// TIA Portal project "TiaUnit" (V16)

(* hardware
DEVICE "S71500/ET200MP-Station_1"  S7-1500 station
   slot 0: "Profilschiene_0"  Rack  6ES7 590-1***0-0AA0
   slot 1: "PLC_1"  CPU 1513-1 PN  6ES7 513-1AL02-0AB0  V2.8
      slot 3: "CPU-Display_1"  6ES7591-1AA00-0AA0
      slot 32768: "PROFINET-Schnittstelle_1"  X1
         slot 32769: "Port_1"  X1 P1
         slot 32770: "Port_2"  X1 P2
      slot 34817: "Virtual CP interface port_1"  Virtual CP interface port  Virtual CP interface port
*)

// ===== PLC "PLC_1"  CPU 1513-1 PN =====

VAR_GLOBAL CONSTANT   // PLC tag table "Assert"
   "NOT_TESTED" : Byte := 16#00;
   "TEST_GOOD" : Byte := 16#01;
   "TEST_BAD" : Byte := 16#02;
END_VAR

TYPE "t_TIAUnit_Tests"
   STRUCT
      "step" : Word;
      result : Byte;
      text : String;
   END_STRUCT;
END_TYPE

TYPE "t_Assert"
   STRUCT
      testStart : Date_And_Time;
      testEnd : Date_And_Time;
      testGood : DInt;
      testBad : DInt;
      index : DInt;
      state : Word;
      stateMachineError : Bool;
   END_STRUCT;
END_TYPE

TYPE "t_AnalogInput"
   STRUCT
      PEW : DInt;   // Peripheral Input
      "Type" : UInt;
      SP1 : Bool;   // Switchpoint 1
      SP2 : Bool;   // Switchpoint 2
      SP3 : Bool;   // Switchpoint 3
      SP4 : Bool;   // Switchpoint 4
      SP5 : Bool;   // Switchpoint 5
      SP6 : Bool;   // Switchpoint 6
      SP7 : Bool;   // Switchpoint 7
      SP8 : Bool;   // Switchpoint 8
      CB : Bool;   // Cable break
      "OF" : Bool;   // Overflow
      SF : Bool;   // Sensor failure
      Bool3 : Bool;
      Bool4 : Bool;
      Bool5 : Bool;
      Bool6 : Bool;
      Bool7 : Bool;
      LoLim : Real := 0.0;   // Scaling Low-Limit
      HiLim : Real := 100.0;   // Scaling High-Limit
      Offset : Real := 0.0;
      Damping : Real := 1.0;   // 0: no damping, damping in s
      ActualValue : Real;   // actual value
      ValueSP1 : Real;   // Value switchpoint 1
      ValueSP2 : Real;   // Value switchpoint 2
      ValueSP3 : Real;   // Value switchpoint 3
      ValueSP4 : Real;   // Value switchpoint 4
      ValueSP5 : Real;   // Value switchpoint 5
      ValueSP6 : Real;   // Value switchpoint 6
      ValueSP7 : Real;   // Value switchpoint 7
      ValueSP8 : Real;   // Value switchpoint 8
      Real9 : Real;
      Real10 : Real;
      Real11 : Real;
      Real12 : Real;
      Real13 : Real;
      Setpoint1 : Real;
      Setpoint2 : Real;
      Setpoint3 : Real;
      Setpoint4 : Real;
      Setpoint5 : Real;
   END_STRUCT;
END_TYPE

DATA_BLOCK "DB_AnalogInput"   // DB4
{ S7_Optimized_Access := 'TRUE' }
VERSION : 0.1
BEGIN
END_DATA_BLOCK

DATA_BLOCK "DB_Simulation"   // DB5
{ S7_Optimized_Access := 'TRUE' }
VERSION : 0.1
   VAR
      value : Real;
      timerOff : IEC_TIMER;
      timerOn : IEC_TIMER;
   END_VAR
BEGIN
END_DATA_BLOCK

DATA_BLOCK "FB_Analogverarbeitung_DB"   // DB6
{ S7_Optimized_Access := 'TRUE' }
VERSION : 0.1
// stored: InstanceOfName FB_Analogverarbeitung
"FB_Analogverarbeitung"
BEGIN
END_DATA_BLOCK

// folder: POUs/TIAUnit_Tests

DATA_BLOCK "FB_Analogverarbeitung_DB_1"   // DB1
{ S7_Optimized_Access := 'TRUE' }
VERSION : 0.1
// stored: InstanceOfName FB_Analogverarbeitung
"FB_Analogverarbeitung"
BEGIN
END_DATA_BLOCK

DATA_BLOCK "FB_Analogverarbeitung_Results"   // DB2
{ S7_Optimized_Access := 'TRUE' }
VERSION : 0.1
   VAR
      Assert : "t_Assert";
      tests : Array[0..100] of "t_TIAUnit_Tests";
   END_VAR
BEGIN
END_DATA_BLOCK

DATA_BLOCK "FB_Analogverarbeitung_Tests_DB"   // DB3
{ S7_Optimized_Access := 'TRUE' }
VERSION : 0.1
// stored: InstanceOfName FB_Analogverarbeitung_Tests
"FB_Analogverarbeitung_Tests"
BEGIN
END_DATA_BLOCK

DATA_BLOCK "DB_AnalogInput_Test"   // DB7
{ S7_Optimized_Access := 'TRUE' }
VERSION : 0.1
BEGIN
END_DATA_BLOCK

// folder: (top level)

FUNCTION_BLOCK "FB_Analogverarbeitung"   // FB1, FBD
{ S7_Optimized_Access := 'TRUE' }
VERSION : 0.1
   VAR_INPUT
      Value : Real;
   END_VAR
   VAR_OUTPUT
      Output : Real;
   END_VAR
   VAR_IN_OUT
      AnalogDB : "t_AnalogInput";
   END_VAR
   VAR
      Filter_PT1_Instance : Filter_PT1;
   END_VAR
   VAR_TEMP
      b_damping : Bool;
      r_input : Real;
      r_value : Real;
   END_VAR
   VAR CONSTANT
      DAMPING_MIN : Real := 0.1;
   END_VAR
BEGIN

REGION Network 1: Limit value
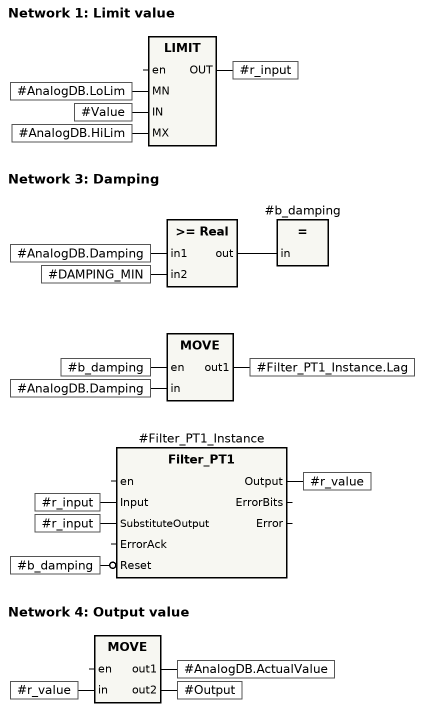
   #r_input := LIMIT(MN := #AnalogDB.LoLim, IN := #Value, MX := #AnalogDB.HiLim);
END_REGION

REGION Network 2 (SCL): Limit setpoints
   #AnalogDB.Setpoint1 := LIMIT(MN := #AnalogDB.LoLim, IN := #AnalogDB.Setpoint1, MX := #AnalogDB.HiLim);
   #AnalogDB.Setpoint2 := LIMIT(MN := #AnalogDB.LoLim, IN := #AnalogDB.Setpoint2, MX := #AnalogDB.HiLim);
   #AnalogDB.Setpoint3 := LIMIT(MN := #AnalogDB.LoLim, IN := #AnalogDB.Setpoint3, MX := #AnalogDB.HiLim);
   #AnalogDB.Setpoint4 := LIMIT(MN := #AnalogDB.LoLim, IN := #AnalogDB.Setpoint4, MX := #AnalogDB.HiLim);
   #AnalogDB.Setpoint5 := LIMIT(MN := #AnalogDB.LoLim, IN := #AnalogDB.Setpoint5, MX := #AnalogDB.HiLim);
END_REGION

REGION Network 3: Damping
   #b_damping := #AnalogDB.Damping >= #DAMPING_MIN;
   IF #b_damping THEN #Filter_PT1_Instance.Lag := #AnalogDB.Damping; END_IF;
   #Filter_PT1_Instance(Input := #r_input,   // Filter_PT1
                        SubstituteOutput := #r_input,
                        Reset := NOT #b_damping,
                        Output => #r_value);
END_REGION

REGION Network 4: Output value
   #AnalogDB.ActualValue := #r_value;
   #Output := #r_value;
END_REGION

REGION Network 5 (SCL): Switchpoints
   #AnalogDB.SP1 := #r_value > #AnalogDB.ValueSP1;
   #AnalogDB.SP2 := #r_value > #AnalogDB.ValueSP2;
   #AnalogDB.SP3 := #r_value > #AnalogDB.ValueSP3;
   #AnalogDB.SP4 := #r_value > #AnalogDB.ValueSP4;
   #AnalogDB.SP5 := #r_value > #AnalogDB.ValueSP5;
   #AnalogDB.SP6 := #r_value > #AnalogDB.ValueSP6;
   #AnalogDB.SP7 := #r_value > #AnalogDB.ValueSP7;
   #AnalogDB.SP8 := #r_value > #AnalogDB.ValueSP8;
END_REGION
END_FUNCTION_BLOCK

ORGANIZATION_BLOCK "Main"   // OB1, FBD, ProgramCycle
TITLE = "Main Program Sweep (Cycle)"
{ S7_Optimized_Access := 'TRUE' }
VERSION : 0.1
   VAR_INPUT
      Initial_Call : Bool;   // Initial call of this OB
      Remanence : Bool;   // =True, if remanent data are available
   END_VAR
   VAR_TEMP
      x_signal : Bool;
      r_value : Real;
      r_dummy : Real;
   END_VAR
BEGIN

REGION Network 1
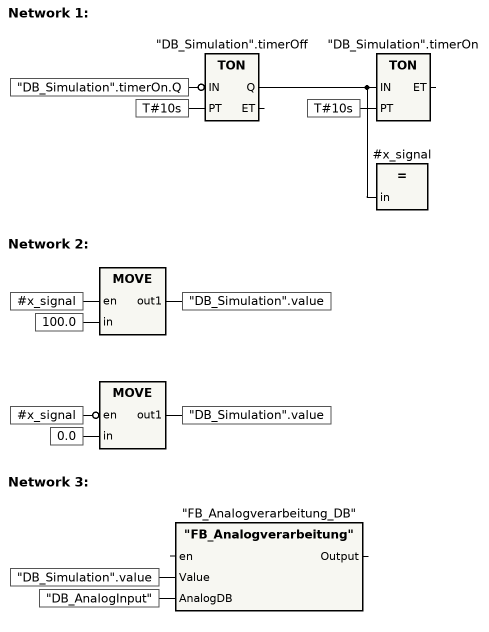
   "DB_Simulation".timerOff.TON(IN := NOT "DB_Simulation".timerOn.Q, PT := T#10s);
   "DB_Simulation".timerOn.TON(IN := "DB_Simulation".timerOff.Q, PT := T#10s);
   #x_signal := "DB_Simulation".timerOff.Q;
END_REGION

REGION Network 2
   IF #x_signal THEN "DB_Simulation".value := 100.0; END_IF;
   IF NOT #x_signal THEN "DB_Simulation".value := 0.0; END_IF;
END_REGION

REGION Network 3
   "FB_Analogverarbeitung_DB"(Value := "DB_Simulation".value, AnalogDB := "DB_AnalogInput");   // "FB_Analogverarbeitung"
END_REGION
END_ORGANIZATION_BLOCK

ORGANIZATION_BLOCK "Programming error"   // OB121, FBD, ProgrammingError
{ S7_Optimized_Access := 'TRUE' }
VERSION : 0.1
   VAR_INPUT
      BlockNr : UInt;   // Number of causing block
      Reaction : USInt;   // 0:ignore, 1:substitute, 2:skip
      Fault_ID : Byte;   // Fault identifier
      BlockType : USInt;   // 16#01:OB, 16#02:FC, 16#03:FB, 16#04:SFC, 16#05:SFB, 16#06:DB: Type of block causing the error
      Area : USInt;   // Area where the error occured
      DBNr : DB_ANY;   // DB number if Area = DB or DI
      Csg_OBNr : OB_Any;   // Number of OB causing the error
      Csg_Prio : USInt;   // Priority of OB causing the error
      Width : USInt;   // 0:bit, 1:byte, 2:word, 3:dword, 4:lword
   END_VAR
BEGIN
END_ORGANIZATION_BLOCK

// folder: POUs/TIAUnit

FUNCTION "Assert_AreEqualREAL" : Void   // FC2, FBD
{ S7_Optimized_Access := 'TRUE' }
VERSION : 0.1
   VAR_INPUT
      Expected : Real;
      Actual : Real;
      Tolerance : Real;
      Message : String;
   END_VAR
   VAR_IN_OUT
      Assert : "t_Assert";
      Test : "t_TIAUnit_Tests";
   END_VAR
   VAR_TEMP
      b_result : Bool;   // Testresult 0: TEST_BAD, 1: TEST_GOOD
      r_hiLim : Real;
      r_loLim : Real;
   END_VAR
BEGIN

REGION Network 1 (SCL): Assert REAL
   #r_hiLim := #Expected + #Tolerance;
   #r_loLim := #Expected - #Tolerance;

   #b_result := FALSE;
   IF #Actual <= #r_hiLim AND #Actual >= #r_loLim THEN
       #b_result := TRUE;
   END_IF;
END_REGION

REGION Network 2: Log Result
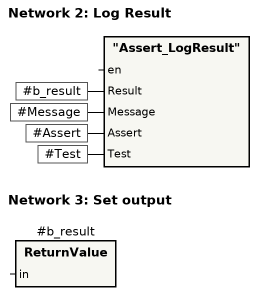
   "Assert_LogResult"(Result := #b_result, Message := #Message, Assert := #Assert, Test := #Test);
END_REGION

REGION Network 3: Set output
   ENO := #b_result;
   RETURN;
END_REGION
END_FUNCTION

FUNCTION "Assert_AreEqualBOOL" : Void   // FC3, FBD
{ S7_Optimized_Access := 'TRUE' }
VERSION : 0.1
   VAR_INPUT
      Expected : Bool;
      Actual : Bool;
      Message : String;
   END_VAR
   VAR_IN_OUT
      Assert : "t_Assert";
      Test : "t_TIAUnit_Tests";
   END_VAR
   VAR_TEMP
      b_result : Bool;   // Testresult 0: TEST_BAD, 1: TEST_GOOD
   END_VAR
BEGIN

REGION Network 1 (SCL): Assert BOOL
   #b_result := FALSE;
   IF #Expected = #Actual THEN
       #b_result := TRUE;
   END_IF;
END_REGION

REGION Network 2: Log Result
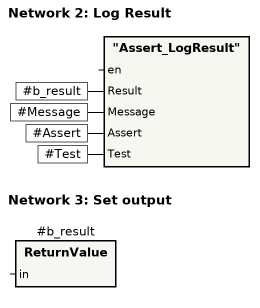
   "Assert_LogResult"(Result := #b_result, Message := #Message, Assert := #Assert, Test := #Test);
END_REGION

REGION Network 3: Set output
   ENO := #b_result;
   RETURN;
END_REGION
END_FUNCTION

FUNCTION "Assert_ClearResults" : Void   // FC4, SCL
{ S7_Optimized_Access := 'TRUE' }
VERSION : 0.1
   VAR_IN_OUT
      Assert : "t_Assert";
      Tests : Array[*] of "t_TIAUnit_Tests";
   END_VAR
   VAR_TEMP
      di_index : DInt;
      i_retVal : Int;
   END_VAR
BEGIN
   REGION Clear assert
       #Assert.index := 0;
       #Assert.stateMachineError := FALSE;
       #i_retVal := RD_SYS_T(#Assert.testStart);
       #Assert.testGood := 0;
       #Assert.testBad := 0;
   END_REGION


   REGION Clear array
       FOR #di_index := LOWER_BOUND(ARR:=#Tests, DIM:=1) TO UPPER_BOUND(ARR:=#Tests, DIM:=1) DO
           #Tests[#di_index].step := 16#0000;
           #Tests[#di_index].result := "NOT_TESTED";
           #Tests[#di_index].text := '';
       END_FOR;
   END_REGION
END_FUNCTION

FUNCTION "Assert_LogResult" : Void   // FC5, SCL
{ S7_Optimized_Access := 'TRUE' }
VERSION : 0.1
   VAR_INPUT
      Result : Bool;
      Message : String;
   END_VAR
   VAR_IN_OUT
      Assert : "t_Assert";
      Test : "t_TIAUnit_Tests";
   END_VAR
   VAR_TEMP
      i_retVal : Int;
      di_length : DInt;
   END_VAR
BEGIN
   REGION #Result
       #Test.step := #Assert.state;
       #Test.text := #Message;
       #Test.result := "TEST_BAD";
       IF (#Result = TRUE) THEN
           #Test.result := "TEST_GOOD";
           #Assert.testGood := #Assert.testGood + 1;
       ELSE
           #Test.result := "TEST_BAD";
           #Assert.testBad := #Assert.testBad + 1;
       END_IF;
       #i_retVal := RD_SYS_T(#Assert.testEnd);
       #Assert.index := #Assert.index + 1;
   END_REGION
END_FUNCTION

FUNCTION "Assert_AreBetweenREAL" : Void   // FC6, FBD
{ S7_Optimized_Access := 'TRUE' }
VERSION : 0.1
   VAR_INPUT
      ExpectedHigh : Real;
      ExpectedLow : Real;
      Actual : Real;
      Tolerance : Real;
      Message : String;
   END_VAR
   VAR_IN_OUT
      Assert : "t_Assert";
      Test : "t_TIAUnit_Tests";
   END_VAR
   VAR_TEMP
      b_result : Bool;   // Testresult 0: TEST_BAD, 1: TEST_GOOD
      r_hiLim : Real;
      r_loLim : Real;
   END_VAR
BEGIN

REGION Network 1 (SCL): Assert REAL
   #r_hiLim := #ExpectedHigh + #Tolerance;
   #r_loLim := #ExpectedLow - #Tolerance;

   #b_result := FALSE;
   IF #Actual >= #r_loLim AND #Actual <= #r_hiLim THEN
       #b_result := TRUE;
   END_IF;
END_REGION

REGION Network 2: Log Result
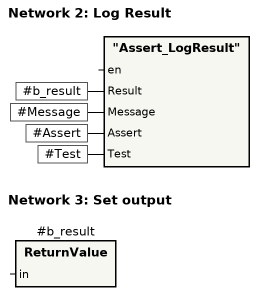
   "Assert_LogResult"(Result := #b_result, Message := #Message, Assert := #Assert, Test := #Test);
END_REGION

REGION Network 3: Set output
   ENO := #b_result;
   RETURN;
END_REGION
END_FUNCTION

// folder: POUs/TIAUnit_Tests

FUNCTION_BLOCK "FB_Analogverarbeitung_Tests"   // FB2, SCL
{ S7_Optimized_Access := 'TRUE' }
VERSION : 0.1
   VAR_OUTPUT
      busy : Bool;
      done : Bool;
      error : Bool;
   END_VAR
   VAR_IN_OUT
      Assert : "t_Assert";
      Tests : Array[*] of "t_TIAUnit_Tests";
   END_VAR
   VAR
      fbTest_0100 : "FB_Analogverarbeitung";
      fbTest_0200 : "FB_Analogverarbeitung";
      fbTest_0300 : "FB_Analogverarbeitung";
      fbTest_0400 : "FB_Analogverarbeitung";
      fbTest_0500 : "FB_Analogverarbeitung";
      fbTest_0600 : "FB_Analogverarbeitung";
      fbTest_0700 : "FB_Analogverarbeitung";
      fbTest_0800 : "FB_Analogverarbeitung";
      fbTest_0900 : "FB_Analogverarbeitung";
      fbTest_1000 : "FB_Analogverarbeitung";
      fbTest_1100 : "FB_Analogverarbeitung";
      fbTest_1200 : "FB_Analogverarbeitung";
      fbTest_1300 : "FB_Analogverarbeitung";
   END_VAR
   VAR_TEMP
      b_result : Bool;
      di_index : DInt;
      r_input : Real;
      r_output : Real;
      r_hiLim : Real;
      r_loLim : Real;
   END_VAR
BEGIN
   CASE #Assert.state OF

       16#0000:  // Initialisation
           #busy := TRUE;
           #done := FALSE;
           #error := FALSE;
           "Assert_ClearResults"(Assert := #Assert, Tests := #Tests);
           "DB_AnalogInput_Test".LoLim := 0.0;
           "DB_AnalogInput_Test".HiLim := 100.0;
           "DB_AnalogInput_Test".Damping := 0.0;
           "DB_AnalogInput_Test".ValueSP1 := 10;
           "DB_AnalogInput_Test".ValueSP2 := 20;
           "DB_AnalogInput_Test".ValueSP3 := 30;
           "DB_AnalogInput_Test".ValueSP4 := 40;
           "DB_AnalogInput_Test".ValueSP5 := 50;
           "DB_AnalogInput_Test".ValueSP6 := 60;
           "DB_AnalogInput_Test".ValueSP7 := 70;
           "DB_AnalogInput_Test".ValueSP8 := 80;
           #Assert.state := 16#0100;


       16#0100:  // Value_ValueBelowLoLim_OutputLo
           #r_input := -10.0;
           #fbTest_0100(Value:=#r_input,
                        AnalogDB:="DB_AnalogInput_Test");
           "Assert_AreEqualREAL"(Expected:="DB_AnalogInput_Test".LoLim,
                                 Actual:="DB_AnalogInput_Test".ActualValue,
                                 Tolerance:=0.1,
                                 Message:='Value_ValueBelowLoLim_OutputLo',
                                 Assert:=#Assert,
                                 Test:=#Tests[#Assert.index]);
           #Assert.state := 16#0200;


       16#0200:  // Value_ValueAboveHiLim_OutputHi
           #r_input := 110.0;
           #fbTest_0200(Value := #r_input,
                        AnalogDB := "DB_AnalogInput_Test");
           "Assert_AreEqualREAL"(Expected := "DB_AnalogInput_Test".HiLim,
                                 Actual := "DB_AnalogInput_Test".ActualValue,
                                 Tolerance := 0.1,
                                 Message := 'Value_ValueAboveHiLim_OutputHi',
                                 Assert := #Assert,
                                 Test := #Tests[#Assert.index]);
           #Assert.state := 16#0300;


       16#0300:  // Value_ValueBetweenLoHi_OutputValue
           #r_input := 60.0;
           #fbTest_0300(Value := #r_input,
                        AnalogDB := "DB_AnalogInput_Test");
           "Assert_AreEqualREAL"(Expected := #r_input,
                                 Actual := "DB_AnalogInput_Test".ActualValue,
                                 Tolerance := 0.1,
                                 Message := 'Value_ValueBetweenLoHi_OutputValue',
                                 Assert := #Assert,
                                 Test := #Tests[#Assert.index]);
           #Assert.state := 16#0400;


       16#0400:  // Value_ValueBelowSP1_AllSPFalse
           #r_input := 5.0;
           #fbTest_0400(Value := #r_input,
                        AnalogDB := "DB_AnalogInput_Test");
           "Assert_AreEqualBOOL"(Expected := FALSE,
                                 Actual := "DB_AnalogInput_Test".SP1,
                                 Message := 'Value_ValueBelowSP1_AllSPFalse',
                                 Assert := #Assert,
                                 Test := #Tests[#Assert.index]);
           "Assert_AreEqualBOOL"(Expected := FALSE,
                                 Actual := "DB_AnalogInput_Test".SP2,
                                 Message := 'Value_ValueBelowSP1_AllSPFalse',
                                 Assert := #Assert,
                                 Test := #Tests[#Assert.index]);
           "Assert_AreEqualBOOL"(Expected := FALSE,
                                 Actual := "DB_AnalogInput_Test".SP3,
                                 Message := 'Value_ValueBelowSP1_AllSPFalse',
                                 Assert := #Assert,
                                 Test := #Tests[#Assert.index]);
           "Assert_AreEqualBOOL"(Expected := FALSE,
                                 Actual := "DB_AnalogInput_Test".SP4,
                                 Message := 'Value_ValueBelowSP1_AllSPFalse',
                                 Assert := #Assert,
                                 Test := #Tests[#Assert.index]);
           "Assert_AreEqualBOOL"(Expected := FALSE,
                                 Actual := "DB_AnalogInput_Test".SP5,
                                 Message := 'Value_ValueBelowSP1_AllSPFalse',
                                 Assert := #Assert,
                                 Test := #Tests[#Assert.index]);
           "Assert_AreEqualBOOL"(Expected := FALSE,
                                 Actual := "DB_AnalogInput_Test".SP6,
                                 Message := 'Value_ValueBelowSP1_AllSPFalse',
                                 Assert := #Assert,
                                 Test := #Tests[#Assert.index]);
           "Assert_AreEqualBOOL"(Expected := FALSE,
                                 Actual := "DB_AnalogInput_Test".SP7,
                                 Message := 'Value_ValueBelowSP1_AllSPFalse',
                                 Assert := #Assert,
                                 Test := #Tests[#Assert.index]);
           "Assert_AreEqualBOOL"(Expected := FALSE,
                                 Actual := "DB_AnalogInput_Test".SP8,
                                 Message := 'Value_ValueBelowSP1_AllSPFalse',
                                 Assert := #Assert,
                                 Test := #Tests[#Assert.index]);
           #Assert.state := 16#0500;


       16#0500:  // Value_ValueBelowSP2_AllSPFalseSP1True
           #r_input := 15.0;
           #fbTest_0500(Value := #r_input,
                        AnalogDB := "DB_AnalogInput_Test");
           "Assert_AreEqualBOOL"(Expected := TRUE,
                                 Actual := "DB_AnalogInput_Test".SP1,
                                 Message := 'Value_ValueBelowSP2_AllSPFalseSP1True',
                                 Assert := #Assert,
                                 Test := #Tests[#Assert.index]);
           "Assert_AreEqualBOOL"(Expected := FALSE,
                                 Actual := "DB_AnalogInput_Test".SP2,
                                 Message := 'Value_ValueBelowSP2_AllSPFalseSP1True',
                                 Assert := #Assert,
                                 Test := #Tests[#Assert.index]);
           "Assert_AreEqualBOOL"(Expected := FALSE,
                                 Actual := "DB_AnalogInput_Test".SP3,
                                 Message := 'Value_ValueBelowSP2_AllSPFalseSP1True',
                                 Assert := #Assert,
                                 Test := #Tests[#Assert.index]);
           "Assert_AreEqualBOOL"(Expected := FALSE,
                                 Actual := "DB_AnalogInput_Test".SP4,
                                 Message := 'Value_ValueBelowSP2_AllSPFalseSP1True',
                                 Assert := #Assert,
                                 Test := #Tests[#Assert.index]);
           "Assert_AreEqualBOOL"(Expected := FALSE,
                                 Actual := "DB_AnalogInput_Test".SP5,
                                 Message := 'Value_ValueBelowSP2_AllSPFalseSP1True',
                                 Assert := #Assert,
                                 Test := #Tests[#Assert.index]);
           "Assert_AreEqualBOOL"(Expected := FALSE,
                                 Actual := "DB_AnalogInput_Test".SP6,
                                 Message := 'Value_ValueBelowSP2_AllSPFalseSP1True',
                                 Assert := #Assert,
                                 Test := #Tests[#Assert.index]);
           "Assert_AreEqualBOOL"(Expected := FALSE,
                                 Actual := "DB_AnalogInput_Test".SP7,
                                 Message := 'Value_ValueBelowSP2_AllSPFalseSP1True',
                                 Assert := #Assert,
                                 Test := #Tests[#Assert.index]);
           "Assert_AreEqualBOOL"(Expected := FALSE,
                                 Actual := "DB_AnalogInput_Test".SP8,
                                 Message := 'Value_ValueBelowSP2_AllSPFalseSP1True',
                                 Assert := #Assert,
                                 Test := #Tests[#Assert.index]);
           #Assert.state := 16#0600;


       16#0600:  // Value_ValueBelowSP3_AllSPFalseSP1and2True
           #r_input := 25.0;
           #fbTest_0600(Value := #r_input,
                        AnalogDB := "DB_AnalogInput_Test");
           "Assert_AreEqualBOOL"(Expected := TRUE,
                                 Actual := "DB_AnalogInput_Test".SP1,
                                 Message := 'Value_ValueBelowSP3_AllSPFalseSP1and2True',
                                 Assert := #Assert,
                                 Test := #Tests[#Assert.index]);
           "Assert_AreEqualBOOL"(Expected := TRUE,
                                 Actual := "DB_AnalogInput_Test".SP2,
                                 Message := 'Value_ValueBelowSP3_AllSPFalseSP1and2True',
                                 Assert := #Assert,
                                 Test := #Tests[#Assert.index]);
           "Assert_AreEqualBOOL"(Expected := FALSE,
                                 Actual := "DB_AnalogInput_Test".SP3,
                                 Message := 'Value_ValueBelowSP3_AllSPFalseSP1and2True',
                                 Assert := #Assert,
                                 Test := #Tests[#Assert.index]);
           "Assert_AreEqualBOOL"(Expected := FALSE,
                                 Actual := "DB_AnalogInput_Test".SP4,
                                 Message := 'Value_ValueBelowSP3_AllSPFalseSP1and2True',
                                 Assert := #Assert,
                                 Test := #Tests[#Assert.index]);
           "Assert_AreEqualBOOL"(Expected := FALSE,
                                 Actual := "DB_AnalogInput_Test".SP5,
                                 Message := 'Value_ValueBelowSP3_AllSPFalseSP1and2True',
                                 Assert := #Assert,
                                 Test := #Tests[#Assert.index]);
           "Assert_AreEqualBOOL"(Expected := FALSE,
                                 Actual := "DB_AnalogInput_Test".SP6,
                                 Message := 'Value_ValueBelowSP3_AllSPFalseSP1and2True',
                                 Assert := #Assert,
                                 Test := #Tests[#Assert.index]);
           "Assert_AreEqualBOOL"(Expected := FALSE,
                                 Actual := "DB_AnalogInput_Test".SP7,
                                 Message := 'Value_ValueBelowSP3_AllSPFalseSP1and2True',
                                 Assert := #Assert,
                                 Test := #Tests[#Assert.index]);
           "Assert_AreEqualBOOL"(Expected := FALSE,
                                 Actual := "DB_AnalogInput_Test".SP8,
                                 Message := 'Value_ValueBelowSP3_AllSPFalseSP1and2True',
                                 Assert := #Assert,
                                 Test := #Tests[#Assert.index]);
           #Assert.state := 16#0700;


       16#0700:  // Value_ValueBelowSP4_AllSPFalseSP12and3True
           #r_input := 35.0;
           #fbTest_0700(Value := #r_input,
                        AnalogDB := "DB_AnalogInput_Test");
           "Assert_AreEqualBOOL"(Expected := TRUE,
                                 Actual := "DB_AnalogInput_Test".SP1,
                                 Message := 'Value_ValueBelowSP4_AllSPFalseSP12and3True',
                                 Assert := #Assert,
                                 Test := #Tests[#Assert.index]);
           "Assert_AreEqualBOOL"(Expected := TRUE,
                                 Actual := "DB_AnalogInput_Test".SP2,
                                 Message := 'Value_ValueBelowSP4_AllSPFalseSP12and3True',
                                 Assert := #Assert,
                                 Test := #Tests[#Assert.index]);
           "Assert_AreEqualBOOL"(Expected := TRUE,
                                 Actual := "DB_AnalogInput_Test".SP3,
                                 Message := 'Value_ValueBelowSP4_AllSPFalseSP12and3True',
                                 Assert := #Assert,
                                 Test := #Tests[#Assert.index]);
           "Assert_AreEqualBOOL"(Expected := FALSE,
                                 Actual := "DB_AnalogInput_Test".SP4,
                                 Message := 'Value_ValueBelowSP4_AllSPFalseSP12and3True',
                                 Assert := #Assert,
                                 Test := #Tests[#Assert.index]);
           "Assert_AreEqualBOOL"(Expected := FALSE,
                                 Actual := "DB_AnalogInput_Test".SP5,
                                 Message := 'Value_ValueBelowSP4_AllSPFalseSP12and3True',
                                 Assert := #Assert,
                                 Test := #Tests[#Assert.index]);
           "Assert_AreEqualBOOL"(Expected := FALSE,
                                 Actual := "DB_AnalogInput_Test".SP6,
                                 Message := 'Value_ValueBelowSP4_AllSPFalseSP12and3True',
                                 Assert := #Assert,
                                 Test := #Tests[#Assert.index]);
           "Assert_AreEqualBOOL"(Expected := FALSE,
                                 Actual := "DB_AnalogInput_Test".SP7,
                                 Message := 'Value_ValueBelowSP4_AllSPFalseSP12and3True',
                                 Assert := #Assert,
                                 Test := #Tests[#Assert.index]);
           "Assert_AreEqualBOOL"(Expected := FALSE,
                                 Actual := "DB_AnalogInput_Test".SP8,
                                 Message := 'Value_ValueBelowSP4_AllSPFalseSP12and3True',
                                 Assert := #Assert,
                                 Test := #Tests[#Assert.index]);
           #Assert.state := 16#0800;


       16#0800:  // Value_ValueBelowSP5_AllSPFalseSP123and4True
           #r_input := 45.0;
           #fbTest_0800(Value := #r_input,
                        AnalogDB := "DB_AnalogInput_Test");
           "Assert_AreEqualBOOL"(Expected := TRUE,
                                 Actual := "DB_AnalogInput_Test".SP1,
                                 Message := 'Value_ValueBelowSP5_AllSPFalseSP123and4True',
                                 Assert := #Assert,
                                 Test := #Tests[#Assert.index]);
           "Assert_AreEqualBOOL"(Expected := TRUE,
                                 Actual := "DB_AnalogInput_Test".SP2,
                                 Message := 'Value_ValueBelowSP5_AllSPFalseSP123and4True',
                                 Assert := #Assert,
                                 Test := #Tests[#Assert.index]);
           "Assert_AreEqualBOOL"(Expected := TRUE,
                                 Actual := "DB_AnalogInput_Test".SP3,
                                 Message := 'Value_ValueBelowSP5_AllSPFalseSP123and4True',
                                 Assert := #Assert,
                                 Test := #Tests[#Assert.index]);
           "Assert_AreEqualBOOL"(Expected := TRUE,
                                 Actual := "DB_AnalogInput_Test".SP4,
                                 Message := 'Value_ValueBelowSP5_AllSPFalseSP123and4True',
                                 Assert := #Assert,
                                 Test := #Tests[#Assert.index]);
           "Assert_AreEqualBOOL"(Expected := FALSE,
                                 Actual := "DB_AnalogInput_Test".SP5,
                                 Message := 'Value_ValueBelowSP5_AllSPFalseSP123and4True',
                                 Assert := #Assert,
                                 Test := #Tests[#Assert.index]);
           "Assert_AreEqualBOOL"(Expected := FALSE,
                                 Actual := "DB_AnalogInput_Test".SP6,
                                 Message := 'Value_ValueBelowSP5_AllSPFalseSP123and4True',
                                 Assert := #Assert,
                                 Test := #Tests[#Assert.index]);
           "Assert_AreEqualBOOL"(Expected := FALSE,
                                 Actual := "DB_AnalogInput_Test".SP7,
                                 Message := 'Value_ValueBelowSP5_AllSPFalseSP123and4True',
                                 Assert := #Assert,
                                 Test := #Tests[#Assert.index]);
           "Assert_AreEqualBOOL"(Expected := FALSE,
                                 Actual := "DB_AnalogInput_Test".SP8,
                                 Message := 'Value_ValueBelowSP5_AllSPFalseSP123and4True',
                                 Assert := #Assert,
                                 Test := #Tests[#Assert.index]);
           #Assert.state := 16#0900;


       16#0900:  // Value_ValueBelowSP6_AllSPFalseSP1234and5True
           #r_input := 55.0;
           #fbTest_0900(Value := #r_input,
                        AnalogDB := "DB_AnalogInput_Test");
           "Assert_AreEqualBOOL"(Expected := TRUE,
                                 Actual := "DB_AnalogInput_Test".SP1,
                                 Message := 'Value_ValueBelowSP6_AllSPFalseSP1234and5True',
                                 Assert := #Assert,
                                 Test := #Tests[#Assert.index]);
           "Assert_AreEqualBOOL"(Expected := TRUE,
                                 Actual := "DB_AnalogInput_Test".SP2,
                                 Message := 'Value_ValueBelowSP6_AllSPFalseSP1234and5True',
                                 Assert := #Assert,
                                 Test := #Tests[#Assert.index]);
           "Assert_AreEqualBOOL"(Expected := TRUE,
                                 Actual := "DB_AnalogInput_Test".SP3,
                                 Message := 'Value_ValueBelowSP6_AllSPFalseSP1234and5True',
                                 Assert := #Assert,
                                 Test := #Tests[#Assert.index]);
           "Assert_AreEqualBOOL"(Expected := TRUE,
                                 Actual := "DB_AnalogInput_Test".SP4,
                                 Message := 'Value_ValueBelowSP6_AllSPFalseSP1234and5True',
                                 Assert := #Assert,
                                 Test := #Tests[#Assert.index]);
           "Assert_AreEqualBOOL"(Expected := TRUE,
                                 Actual := "DB_AnalogInput_Test".SP5,
                                 Message := 'Value_ValueBelowSP6_AllSPFalseSP1234and5True',
                                 Assert := #Assert,
                                 Test := #Tests[#Assert.index]);
           "Assert_AreEqualBOOL"(Expected := FALSE,
                                 Actual := "DB_AnalogInput_Test".SP6,
                                 Message := 'Value_ValueBelowSP6_AllSPFalseSP1234and5True',
                                 Assert := #Assert,
                                 Test := #Tests[#Assert.index]);
           "Assert_AreEqualBOOL"(Expected := FALSE,
                                 Actual := "DB_AnalogInput_Test".SP7,
                                 Message := 'Value_ValueBelowSP6_AllSPFalseSP1234and5True',
                                 Assert := #Assert,
                                 Test := #Tests[#Assert.index]);
           "Assert_AreEqualBOOL"(Expected := FALSE,
                                 Actual := "DB_AnalogInput_Test".SP8,
                                 Message := 'Value_ValueBelowSP6_AllSPFalseSP1234and5True',
                                 Assert := #Assert,
                                 Test := #Tests[#Assert.index]);
           #Assert.state := 16#1000;


       16#1000:  // Value_ValueBelowSP7_AllSPFalseSP12345and6True
           #r_input := 65.0;
           #fbTest_1000(Value := #r_input,
                        AnalogDB := "DB_AnalogInput_Test");
           "Assert_AreEqualBOOL"(Expected := TRUE,
                                 Actual := "DB_AnalogInput_Test".SP1,
                                 Message := 'Value_ValueBelowSP7_AllSPFalseSP12345and6True',
                                 Assert := #Assert,
                                 Test := #Tests[#Assert.index]);
           "Assert_AreEqualBOOL"(Expected := TRUE,
                                 Actual := "DB_AnalogInput_Test".SP2,
                                 Message := 'Value_ValueBelowSP7_AllSPFalseSP12345and6True',
                                 Assert := #Assert,
                                 Test := #Tests[#Assert.index]);
           "Assert_AreEqualBOOL"(Expected := TRUE,
                                 Actual := "DB_AnalogInput_Test".SP3,
                                 Message := 'Value_ValueBelowSP7_AllSPFalseSP12345and6True',
                                 Assert := #Assert,
                                 Test := #Tests[#Assert.index]);
           "Assert_AreEqualBOOL"(Expected := TRUE,
                                 Actual := "DB_AnalogInput_Test".SP4,
                                 Message := 'Value_ValueBelowSP7_AllSPFalseSP12345and6True',
                                 Assert := #Assert,
                                 Test := #Tests[#Assert.index]);
           "Assert_AreEqualBOOL"(Expected := TRUE,
                                 Actual := "DB_AnalogInput_Test".SP5,
                                 Message := 'Value_ValueBelowSP7_AllSPFalseSP12345and6True',
                                 Assert := #Assert,
                                 Test := #Tests[#Assert.index]);
           "Assert_AreEqualBOOL"(Expected := TRUE,
                                 Actual := "DB_AnalogInput_Test".SP6,
                                 Message := 'Value_ValueBelowSP7_AllSPFalseSP12345and6True',
                                 Assert := #Assert,
                                 Test := #Tests[#Assert.index]);
           "Assert_AreEqualBOOL"(Expected := FALSE,
                                 Actual := "DB_AnalogInput_Test".SP7,
                                 Message := 'Value_ValueBelowSP7_AllSPFalseSP12345and6True',
                                 Assert := #Assert,
                                 Test := #Tests[#Assert.index]);
           "Assert_AreEqualBOOL"(Expected := FALSE,
                                 Actual := "DB_AnalogInput_Test".SP8,
                                 Message := 'Value_ValueBelowSP7_AllSPFalseSP12345and6True',
                                 Assert := #Assert,
                                 Test := #Tests[#Assert.index]);
           #Assert.state := 16#1100;


       16#1100:  // Value_ValueBelowSP8_AllSPFalseSP123456and7True
           #r_input := 75.0;
           #fbTest_1100(Value := #r_input,
                        AnalogDB := "DB_AnalogInput_Test");
           "Assert_AreEqualBOOL"(Expected := TRUE,
                                 Actual := "DB_AnalogInput_Test".SP1,
                                 Message := 'Value_ValueBelowSP8_AllSPFalseSP123456and7True',
                                 Assert := #Assert,
                                 Test := #Tests[#Assert.index]);
           "Assert_AreEqualBOOL"(Expected := TRUE,
                                 Actual := "DB_AnalogInput_Test".SP2,
                                 Message := 'Value_ValueBelowSP8_AllSPFalseSP123456and7True',
                                 Assert := #Assert,
                                 Test := #Tests[#Assert.index]);
           "Assert_AreEqualBOOL"(Expected := TRUE,
                                 Actual := "DB_AnalogInput_Test".SP3,
                                 Message := 'Value_ValueBelowSP8_AllSPFalseSP123456and7True',
                                 Assert := #Assert,
                                 Test := #Tests[#Assert.index]);
           "Assert_AreEqualBOOL"(Expected := TRUE,
                                 Actual := "DB_AnalogInput_Test".SP4,
                                 Message := 'Value_ValueBelowSP8_AllSPFalseSP123456and7True',
                                 Assert := #Assert,
                                 Test := #Tests[#Assert.index]);
           "Assert_AreEqualBOOL"(Expected := TRUE,
                                 Actual := "DB_AnalogInput_Test".SP5,
                                 Message := 'Value_ValueBelowSP8_AllSPFalseSP123456and7True',
                                 Assert := #Assert,
                                 Test := #Tests[#Assert.index]);
           "Assert_AreEqualBOOL"(Expected := TRUE,
                                 Actual := "DB_AnalogInput_Test".SP6,
                                 Message := 'Value_ValueBelowSP8_AllSPFalseSP123456and7True',
                                 Assert := #Assert,
                                 Test := #Tests[#Assert.index]);
           "Assert_AreEqualBOOL"(Expected := TRUE,
                                 Actual := "DB_AnalogInput_Test".SP7,
                                 Message := 'Value_ValueBelowSP8_AllSPFalseSP123456and7True',
                                 Assert := #Assert,
                                 Test := #Tests[#Assert.index]);
           "Assert_AreEqualBOOL"(Expected := FALSE,
                                 Actual := "DB_AnalogInput_Test".SP8,
                                 Message := 'Value_ValueBelowSP8_AllSPFalseSP123456and7True',
                                 Assert := #Assert,
                                 Test := #Tests[#Assert.index]);
           #Assert.state := 16#1200;


       16#1200:  // Value_ValueAbovewSP8_AllSPTrue
           #r_input := 85.0;
           #fbTest_1200(Value := #r_input,
                        AnalogDB := "DB_AnalogInput_Test");
           "Assert_AreEqualBOOL"(Expected := TRUE,
                                 Actual := "DB_AnalogInput_Test".SP1,
                                 Message := 'Value_ValueAbovewSP8_AllSPTrue',
                                 Assert := #Assert,
                                 Test := #Tests[#Assert.index]);
           "Assert_AreEqualBOOL"(Expected := TRUE,
                                 Actual := "DB_AnalogInput_Test".SP2,
                                 Message := 'Value_ValueAbovewSP8_AllSPTrue',
                                 Assert := #Assert,
                                 Test := #Tests[#Assert.index]);
           "Assert_AreEqualBOOL"(Expected := TRUE,
                                 Actual := "DB_AnalogInput_Test".SP3,
                                 Message := 'Value_ValueAbovewSP8_AllSPTrue',
                                 Assert := #Assert,
                                 Test := #Tests[#Assert.index]);
           "Assert_AreEqualBOOL"(Expected := TRUE,
                                 Actual := "DB_AnalogInput_Test".SP4,
                                 Message := 'Value_ValueAbovewSP8_AllSPTrue',
                                 Assert := #Assert,
                                 Test := #Tests[#Assert.index]);
           "Assert_AreEqualBOOL"(Expected := TRUE,
                                 Actual := "DB_AnalogInput_Test".SP5,
                                 Message := 'Value_ValueAbovewSP8_AllSPTrue',
                                 Assert := #Assert,
                                 Test := #Tests[#Assert.index]);
           "Assert_AreEqualBOOL"(Expected := TRUE,
                                 Actual := "DB_AnalogInput_Test".SP6,
                                 Message := 'Value_ValueAbovewSP8_AllSPTrue',
                                 Assert := #Assert,
                                 Test := #Tests[#Assert.index]);
           "Assert_AreEqualBOOL"(Expected := TRUE,
                                 Actual := "DB_AnalogInput_Test".SP7,
                                 Message := 'Value_ValueAbovewSP8_AllSPTrue',
                                 Assert := #Assert,
                                 Test := #Tests[#Assert.index]);
           "Assert_AreEqualBOOL"(Expected := TRUE,
                                 Actual := "DB_AnalogInput_Test".SP8,
                                 Message := 'Value_ValueAbovewSP8_AllSPTrue',
                                 Assert := #Assert,
                                 Test := #Tests[#Assert.index]);
           #Assert.state := 16#1300;


       16#1300:  // Setpoints_ValueBelowOrAboveLimits_SetpointsBetweenLoAndHi
           #r_input := 85.0;
           "DB_AnalogInput_Test".Setpoint1 := -10.0;
           "DB_AnalogInput_Test".Setpoint2 := 110.0;
           "DB_AnalogInput_Test".Setpoint3 := -20.0;
           "DB_AnalogInput_Test".Setpoint4 := 210.0;
           "DB_AnalogInput_Test".Setpoint5 := -10.0;
           #fbTest_1300(Value := #r_input,
                        AnalogDB := "DB_AnalogInput_Test");
           "Assert_AreBetweenREAL"(ExpectedHigh := "DB_AnalogInput_Test".HiLim,
                                   ExpectedLow := "DB_AnalogInput_Test".LoLim,
                                   Actual := "DB_AnalogInput_Test".Setpoint1,
                                   Tolerance := 0.1,
                                   Message := 'Setpoints_ValueBelowOrAboveLimits_SetpointsBetweenLoAndHi',
                                   Assert := #Assert,
                                   Test := #Tests[#Assert.index]);
           "Assert_AreBetweenREAL"(ExpectedHigh := "DB_AnalogInput_Test".HiLim,
                                   ExpectedLow := "DB_AnalogInput_Test".LoLim,
                                   Actual := "DB_AnalogInput_Test".Setpoint2,
                                   Tolerance := 0.1,
                                   Message := 'Setpoints_ValueBelowOrAboveLimits_SetpointsBetweenLoAndHi',
                                   Assert := #Assert,
                                   Test := #Tests[#Assert.index]);
           "Assert_AreBetweenREAL"(ExpectedHigh := "DB_AnalogInput_Test".HiLim,
                                   ExpectedLow := "DB_AnalogInput_Test".LoLim,
                                   Actual := "DB_AnalogInput_Test".Setpoint3,
                                   Tolerance := 0.1,
                                   Message := 'Setpoints_ValueBelowOrAboveLimits_SetpointsBetweenLoAndHi',
                                   Assert := #Assert,
                                   Test := #Tests[#Assert.index]);
           "Assert_AreBetweenREAL"(ExpectedHigh := "DB_AnalogInput_Test".HiLim,
                                   ExpectedLow := "DB_AnalogInput_Test".LoLim,
                                   Actual := "DB_AnalogInput_Test".Setpoint4,
                                   Tolerance := 0.1,
                                   Message := 'Setpoints_ValueBelowOrAboveLimits_SetpointsBetweenLoAndHi',
                                   Assert := #Assert,
                                   Test := #Tests[#Assert.index]);
           "Assert_AreBetweenREAL"(ExpectedHigh := "DB_AnalogInput_Test".HiLim,
                                   ExpectedLow := "DB_AnalogInput_Test".LoLim,
                                   Actual := "DB_AnalogInput_Test".Setpoint5,
                                   Tolerance := 0.1,
                                   Message := 'Setpoints_ValueBelowOrAboveLimits_SetpointsBetweenLoAndHi',
                                   Assert := #Assert,
                                   Test := #Tests[#Assert.index]);
           #Assert.state := 16#FF00;



       16#FF00:  // done
           #busy := FALSE;
           #done := TRUE;


       16#FFFF:   // Error
           #busy := FALSE;
           #error := TRUE;


       ELSE  // Statement section ELSE
           #Assert.stateMachineError := True;
   END_CASE;
END_FUNCTION_BLOCK

ORGANIZATION_BLOCK "P_Unit_Tests"   // OB123, FBD, ProgramCycle
TITLE = "Main Program Sweep (Cycle)"
{ S7_Optimized_Access := 'TRUE' }
VERSION : 0.1
   VAR_INPUT
      Initial_Call : Bool;   // Initial call of this OB
      Remanence : Bool;   // =True, if remanent data are available
   END_VAR
BEGIN

REGION Network 1
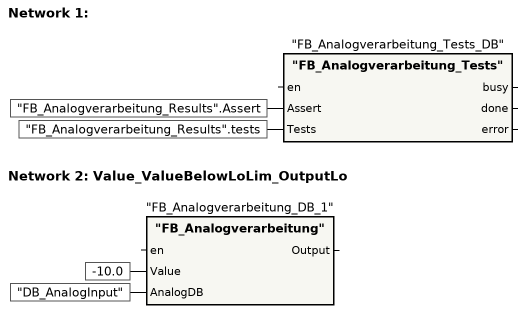
   "FB_Analogverarbeitung_Tests_DB"(Assert := "FB_Analogverarbeitung_Results".Assert,   // "FB_Analogverarbeitung_Tests"
                           Tests := "FB_Analogverarbeitung_Results".tests);
END_REGION

REGION Network 2: Value_ValueBelowLoLim_OutputLo
   "FB_Analogverarbeitung_DB_1"(Value := -10.0, AnalogDB := "DB_AnalogInput");   // "FB_Analogverarbeitung"
END_REGION
END_ORGANIZATION_BLOCK